Fanuc KAREL source: compact_preamble.KL

PROGRAM KB00020
%NOLOCKGROUP
VAR
P1:INTEGER;RESULT : STRING[80]
BEGIN
P1=1
RESULT=CHR(P1)
END KB00020
